TYPE ST_ErrorSource :
STRUCT
	InstanceName	: Tc2_System.T_MaxString;
	ErrorCode		: DINT;
	Description		: Tc2_System.T_MaxString;
END_STRUCT
END_TYPE

(* stored: Version 1.1.0.1, ProductVersion 3.1.4024.13
   DUT ST_ErrorSource: Id {82858906-bd52-094e-0b2f-0b5b1d45ef8f} *)
